{attribute 'qualified_only'}
TYPE E_PulseOptions :
(
	Off :=16#00,
    FadeBlue :=16#01,
    FadeOut :=16#02
) INT;
END_TYPE

(* stored: Version 1.1.0.1, ProductVersion 3.1.4024.9
   DUT E_PulseOptions: Id {c0a4182a-168d-44f1-8e86-ff1e20bc5a5d} *)
